// TwinCAT 3 PLC project PLC
// ProgramVersion: 3.1.4024.0
// libraries:
//   SPT Base Types, * (Beckhoff Automation LLC)
//   Tc2_Standard, * (Beckhoff Automation GmbH)
//   Tc2_System, * (Beckhoff Automation GmbH)
//   Tc3_Module, * (Beckhoff Automation GmbH)
//   Tc3_PackML_V2, * (Beckhoff Automation GmbH)
//   VisuDialogs, * (System)
// project tree:
//   DUTs/HMI/ ST_HMI_Machine.TcDUT, ST_HMI_Machine_Command.TcDUT, ST_HMI_Machine_Config.TcDUT, ST_HMI_Machine_Status.TcDUT
//   / GlobalTextList.TcGTLO, PlcTask.TcTTO, Visualization Manager.TcVMO (not stored)
//   POUs/ MAIN.TcPOU
//   VISUs/VFMs/ VFM_Machine.TcVIS, VFM_MachineControl.TcVIS, VFM_Module.TcVIS, VFM_OperatingMode.TcVIS, VFM_PackML.TcVIS, VFM_PackML_Manual.TcVIS
//   VISUs/ VIS_Main.TcVIS, VIS_TempCtrl.TcVIS
//   _Machine/00_Machine/ FB_UM_Machine.TcPOU
//   _Machine/_Components/Misc/ FB_StatFilter.TcPOU, FB_TempCtrl.TcPOU, F_TaskTime.TcPOU
//   _Machine/_Components/TempController/DUTs/ ST_HMI_TempController.TcDUT, ST_HMI_TempController_Command.TcDUT, ST_HMI_TempController_Config.TcDUT, ST_HMI_TempController_Status.TcDUT, ST_Param_TempController.TcDUT
//   _Machine/_Components/TempController/ FB_TempController.TcPOU, I_TemperatureController.TcIO
//   _Machine/_Components/TempController/VFMs/ VFM_TempController.TcVIS
// real-time tasks:
//   TASK PlcTask: cycle T#10ms, priority 20, ADS port 350

CONFIGURATION PLC
    RESOURCE PLC ON TwinCAT3
        TASK PlcTask(INTERVAL := T#10ms, PRIORITY := 20);
        PROGRAM MAIN WITH PlcTask : MAIN;
    END_RESOURCE
END_CONFIGURATION

// ---- DUTs/HMI/ST_HMI_Machine.TcDUT
TYPE ST_HMI_Machine :
STRUCT
	Command: ST_HMI_Machine_Command;
	Config: ST_HMI_Machine_Config;
	Status: ST_HMI_Machine_Status;
END_STRUCT
END_TYPE

// ---- DUTs/HMI/ST_HMI_Machine_Command.TcDUT
TYPE ST_HMI_Machine_Command :
STRUCT
	Start: BOOL;
	Stop: BOOL;
	Reset: BOOL;
	Abort: BOOL;
END_STRUCT
END_TYPE

// ---- DUTs/HMI/ST_HMI_Machine_Config.TcDUT
TYPE ST_HMI_Machine_Config :
STRUCT
END_STRUCT
END_TYPE

// ---- DUTs/HMI/ST_HMI_Machine_Status.TcDUT
TYPE ST_HMI_Machine_Status :
STRUCT
END_STRUCT
END_TYPE

// ---- _Machine/_Components/TempController/DUTs/ST_HMI_TempController.TcDUT
TYPE ST_HMI_TempController :
STRUCT
	Command: ST_HMI_TempController_Command;
	Config: ST_HMI_TempController_Config;
	Status: ST_HMI_TempController_Status;
END_STRUCT
END_TYPE

// ---- _Machine/_Components/TempController/DUTs/ST_HMI_TempController_Command.TcDUT
TYPE ST_HMI_TempController_Command :
STRUCT
	Manual: BOOL := TRUE;
	Start: BOOL;
	Stop: BOOL;
	ResetPID: BOOL;
END_STRUCT
END_TYPE

// ---- _Machine/_Components/TempController/DUTs/ST_HMI_TempController_Config.TcDUT
TYPE ST_HMI_TempController_Config :
STRUCT
	Param: ST_Param_TempController;
END_STRUCT
END_TYPE

// ---- _Machine/_Components/TempController/DUTs/ST_HMI_TempController_Status.TcDUT
TYPE ST_HMI_TempController_Status :
STRUCT
	Enabled: BOOL;
	CtrlOutput: LREAL;
	Actual: LREAL;
END_STRUCT
END_TYPE

// ---- _Machine/_Components/TempController/DUTs/ST_Param_TempController.TcDUT
TYPE ST_Param_TempController :
STRUCT
	MaxTemp: LREAL := 350.0;
	Setpoint: LREAL := 20.0;
	Range: LREAL := 10.0;
	Kp: LREAL := 1.0;
	Tn: LREAL := 0.005;
	Tv: LREAL := 0.0;
	Td: LREAL := 0.0;
END_STRUCT
END_TYPE

// ---- _Machine/_Components/TempController/I_TemperatureController.TcIO
INTERFACE I_TemperatureController

METHOD Disable
VAR_INPUT
END_VAR
END_METHOD

METHOD Enable
VAR_INPUT
END_VAR
END_METHOD

PROPERTY Enabled : bool
GET
END_GET
END_PROPERTY

END_INTERFACE

// ---- POUs/MAIN.TcPOU
(*	Sample Code Disclaimer
	All sample code provided by Beckhoff Automation LLC are for illustrative purposes only
	and are provided “as is” and without any warranties, express or implied.
	Actual implementations in applications will vary significantly.
	Beckhoff Automation LLC shall have no liability for, and does not waive any rights in relation to,
	any code samples that it provides or the use of such code samples for any purpose.
*)
PROGRAM MAIN
VAR
	Machine: FB_UM_Machine	:= (Name := 'Machine', LogStateChanges := TRUE);
	Initialized: BOOL;
END_VAR

CyclicLogic();

METHOD CyclicLogic : BOOL
VAR_INPUT
END_VAR
IF NOT Initialized THEN
    Initialized := Initialize();
    RETURN;
END_IF

Machine.CyclicLogic();
END_METHOD

METHOD Initialize : BOOL
VAR_INPUT
END_VAR
Initialize := TRUE;
END_METHOD

END_PROGRAM

// ---- _Machine/00_Machine/FB_UM_Machine.TcPOU
FUNCTION_BLOCK FB_UM_Machine EXTENDS FB_PackML_BaseModule
VAR
	// Submodules
	
	// Components
	TempController: FB_TempController	:= (Name := 'Temperature Controller');
	
	// Module Data
	// --Param
	// --Recipe
	// --HMI
	HMI: ST_HMI_Machine;
	
	// Alarms
	
	// Other I/O

	// Machine Control
	rtrigControl: R_TRIG;
	CheckAbort: BOOL;
	CheckStop: BOOL;
	
	// Miscellaneous
	
END_VAR

METHOD PROTECTED Aborted
VAR_INPUT
END_VAR
END_METHOD

METHOD PROTECTED Aborting
VAR_INPUT
END_VAR
CASE _CurrentMode OF
	E_PMLUnitMode.ePMLUnitMode_Production:
        CASE DescendantSequenceState OF
			0:
				NoStateTasksToComplete := FALSE;
				DescendantSequenceState := DescendantSequenceState + 10;
			10:
				StateTasksComplete := TRUE;
		END_CASE
		
	E_PMLUnitMode.ePMLUnitMode_Manual, E_PMLUnitMode.ePMLUnitMode_Maintenance:
        ;	
END_CASE

// Call Super
SUPER^.Aborting();
END_METHOD

METHOD PROTECTED Clearing
VAR_INPUT
END_VAR
CASE _CurrentMode OF
	E_PMLUnitMode.ePMLUnitMode_Production:
        CASE DescendantSequenceState OF
			0:
				NoStateTasksToComplete := FALSE;
				DescendantSequenceState := DescendantSequenceState + 10;
			10:
				StateTasksComplete := TRUE;
		END_CASE
		
	E_PMLUnitMode.ePMLUnitMode_Manual, E_PMLUnitMode.ePMLUnitMode_Maintenance:
        ;	
END_CASE

// Call Super
SUPER^.Clearing();
END_METHOD

METHOD PROTECTED Complete
VAR_INPUT
END_VAR
END_METHOD

//! @summary Initializes event function blocks using this module's name
METHOD PROTECTED CreateEvents

//! @description This method is called by <c>Initialize()</c> as required
// Add your event creation here

// Super call to base
SUPER^.CreateEvents();
END_METHOD

METHOD CyclicLogic
VAR_INPUT
END_VAR
IF NOT _InitComplete THEN
    _InitComplete := Initialize();
    RETURN;
END_IF

MachineControl();

SUPER^.CyclicLogic();
END_METHOD

METHOD PROTECTED Execute
VAR_INPUT
END_VAR
CASE _CurrentMode OF
	E_PMLUnitMode.ePMLUnitMode_Production:
        CASE DescendantSequenceState OF
			0:
				DescendantSequenceState := DescendantSequenceState + 10;
			10:
				;
		END_CASE
		
	E_PMLUnitMode.ePMLUnitMode_Manual, E_PMLUnitMode.ePMLUnitMode_Maintenance:
        ;	
END_CASE
END_METHOD

METHOD PROTECTED Held
VAR_INPUT
END_VAR
END_METHOD

METHOD PROTECTED Holding
VAR_INPUT
END_VAR
CASE _CurrentMode OF
	E_PMLUnitMode.ePMLUnitMode_Production:
        CASE DescendantSequenceState OF
			0:
				NoStateTasksToComplete := FALSE;
				DescendantSequenceState := DescendantSequenceState + 10;
			10:
				StateTasksComplete := TRUE;
		END_CASE
		
	E_PMLUnitMode.ePMLUnitMode_Manual, E_PMLUnitMode.ePMLUnitMode_Maintenance:
        ;	
END_CASE

// Call Super
SUPER^.Holding();
END_METHOD

METHOD PROTECTED Idle
VAR_INPUT
END_VAR
END_METHOD

//! @summary Basic module initialization logic
METHOD PROTECTED Initialize : BOOL;
VAR
	i						 : UDINT;
	varInfo					 : __SYSTEM.VAR_INFO;
	AllSubUnitsInitialized	 : BOOL := TRUE;
	AllComponentsInitialized : BOOL := TRUE;
END_VAR

//! @description This method is called by <c>CyclicLogic()</c> as required
Initialize := FALSE;
CASE DescendantSequenceState OF
    0: // Initialize
        _LogModeChanges         := FALSE;
        _LogStateChanges        := FALSE;
        DescendantSequenceState := DescendantSequenceState + 10;
	
	10: // Register Submodules
		DescendantSequenceState := DescendantSequenceState + 10;
		
    20: // Register Components
		RegisterComponent(TempController);
        DescendantSequenceState := DescendantSequenceState + 10;
		
    30: // Call the Super
        IF SUPER^.Initialize() THEN
            DescendantSequenceState := DescendantSequenceState + 10;
        END_IF
    40:
        Initialize := TRUE;
END_CASE
END_METHOD

METHOD MachineControl
VAR_INPUT
END_VAR
// Control Triggers
rtrigControl(CLK:= HMI.Command.Start XOR HMI.Command.Stop XOR HMI.Command.Reset XOR HMI.Command.Abort);

CASE CurrentState OF
	E_PMLState.ePMLState_Aborting:
		CheckAbort := FALSE;
		CheckStop := FALSE;
		
	E_PMLState.ePMLState_Aborted:
		// Wait for Reset to Clear
		IF rtrigControl.Q AND HMI.Command.Reset THEN
			ChangeState(E_PMLCommand.ePMLCommand_Clear);
		END_IF
		
	E_PMLState.ePMLState_Clearing:
		CheckAbort := TRUE;
		CheckStop := FALSE;
		
	E_PMLState.ePMLState_Stopping:
		CheckAbort := TRUE;
		CheckStop := FALSE;
		
	E_PMLState.ePMLState_Stopped:
		// Wait for Reset
		IF rtrigControl.Q AND HMI.Command.Reset THEN
			ChangeState(E_PMLCommand.ePMLCommand_Reset);
		END_IF
		
	E_PMLState.ePMLState_Resetting:
		CheckAbort := TRUE;
		CheckStop := TRUE;
	
	E_PMLState.ePMLState_Idle:
		// Wait for Start
		IF rtrigControl.Q AND HMI.Command.Start THEN
			ChangeState(E_PMLCommand.ePMLCommand_Start);
		END_IF
	
END_CASE

// Check for Abort or Stop
IF rtrigControl.Q AND HMI.Command.Abort THEN
	ChangeState(E_PMLCommand.ePMLCommand_Abort);
ELSIF rtrigControl.Q AND HMI.Command.Stop THEN
	ChangeState(E_PMLCommand.ePMLCommand_Stop);
END_IF
END_METHOD

METHOD PROTECTED Resetting
VAR_INPUT
END_VAR
CASE _CurrentMode OF
	E_PMLUnitMode.ePMLUnitMode_Production:
        CASE DescendantSequenceState OF
			0:
				NoStateTasksToComplete := FALSE;
				DescendantSequenceState := DescendantSequenceState + 10;
			10:
				StateTasksComplete := TRUE;
		END_CASE
		
	E_PMLUnitMode.ePMLUnitMode_Manual, E_PMLUnitMode.ePMLUnitMode_Maintenance:
        ;	
END_CASE

// Call Super
SUPER^.Resetting();
END_METHOD

METHOD PROTECTED Starting
VAR_INPUT
END_VAR
CASE _CurrentMode OF
	E_PMLUnitMode.ePMLUnitMode_Production:
        CASE DescendantSequenceState OF
			0:
				NoStateTasksToComplete := FALSE;
				DescendantSequenceState := DescendantSequenceState + 10;
			10:
				StateTasksComplete := TRUE;
		END_CASE
		
	E_PMLUnitMode.ePMLUnitMode_Manual, E_PMLUnitMode.ePMLUnitMode_Maintenance:
        ;	
END_CASE

// Call Super
SUPER^.Starting();
END_METHOD

METHOD PROTECTED Stopped
VAR_INPUT
END_VAR
END_METHOD

METHOD PROTECTED Stopping
VAR_INPUT
END_VAR
CASE _CurrentMode OF
	E_PMLUnitMode.ePMLUnitMode_Production:
        CASE DescendantSequenceState OF
			0:
				NoStateTasksToComplete := FALSE;
				DescendantSequenceState := DescendantSequenceState + 10;
			10:
				StateTasksComplete := TRUE;
		END_CASE
		
	E_PMLUnitMode.ePMLUnitMode_Manual, E_PMLUnitMode.ePMLUnitMode_Maintenance:
        ;	
END_CASE

// Call Super
SUPER^.Stopping();
END_METHOD

METHOD PROTECTED Suspended
VAR_INPUT
END_VAR
END_METHOD

METHOD PROTECTED Suspending
VAR_INPUT
END_VAR
CASE _CurrentMode OF
	E_PMLUnitMode.ePMLUnitMode_Production:
        CASE DescendantSequenceState OF
			0:
				NoStateTasksToComplete := FALSE;
				DescendantSequenceState := DescendantSequenceState + 10;
			10:
				StateTasksComplete := TRUE;
		END_CASE
		
	E_PMLUnitMode.ePMLUnitMode_Manual, E_PMLUnitMode.ePMLUnitMode_Maintenance:
        ;	
END_CASE

// Call Super
SUPER^.Suspending();
END_METHOD

METHOD PROTECTED Undefined
VAR_INPUT
END_VAR
END_METHOD

METHOD PROTECTED Unholding
VAR_INPUT
END_VAR
CASE _CurrentMode OF
	E_PMLUnitMode.ePMLUnitMode_Production:
        CASE DescendantSequenceState OF
			0:
				NoStateTasksToComplete := FALSE;
				DescendantSequenceState := DescendantSequenceState + 10;
			10:
				StateTasksComplete := TRUE;
		END_CASE
		
	E_PMLUnitMode.ePMLUnitMode_Manual, E_PMLUnitMode.ePMLUnitMode_Maintenance:
        ;	
END_CASE

// Call Super
SUPER^.Unholding();
END_METHOD

METHOD PROTECTED Unsuspending
VAR_INPUT
END_VAR
CASE _CurrentMode OF
	E_PMLUnitMode.ePMLUnitMode_Production:
        CASE DescendantSequenceState OF
			0:
				NoStateTasksToComplete := FALSE;
				DescendantSequenceState := DescendantSequenceState + 10;
			10:
				StateTasksComplete := TRUE;
		END_CASE
		
	E_PMLUnitMode.ePMLUnitMode_Manual, E_PMLUnitMode.ePMLUnitMode_Maintenance:
        ;	
END_CASE

// Call Super
SUPER^.Unsuspending();
END_METHOD

END_FUNCTION_BLOCK

// ---- _Machine/_Components/TempController/FB_TempController.TcPOU
(*	Sample Code Disclaimer
	All sample code provided by Beckhoff Automation LLC are for illustrative purposes only
	and are provided “as is” and without any warranties, express or implied.
	Actual implementations in applications will vary significantly.
	Beckhoff Automation LLC shall have no liability for, and does not waive any rights in relation to,
	any code samples that it provides or the use of such code samples for any purpose.
*)
FUNCTION_BLOCK FB_TempController EXTENDS FB_ComponentBase IMPLEMENTS I_TemperatureController
VAR	
	// Properties
	_Enabled: BOOL;
		
	// HMI Interface
	HMI: ST_HMI_TempController;
	
	// Hardware Inputs
	//Feedback AT %I*: INT;
	
	// Hardware Outputs
	CtrlOut AT %Q*: INT; // Scaled for HW Output

	// General
	fbTempCtrl: FB_TempCtrl;
	Setpoint: LREAL;
	Feedback: LREAL; // Scaled for HW Input
	ResetPID: BOOL;
	PID_Output: LREAL;
	EnableReq: BOOL;
	DisableReq: BOOL;
	
	// Simulation

END_VAR

VAR PERSISTENT
	Param: ST_Param_TempController;
END_VAR

METHOD CyclicLogic
VAR_INPUT
END_VAR
// Call Super
SUPER^.CyclicLogic();

IF EnableReq THEN
	_Enabled := TRUE;
	EnableReq := FALSE;
ELSIF DisableReq OR Feedback >= Param.MaxTemp THEN
	_Enabled := FALSE;	
	DisableReq := FALSE;
END_IF

// Input Scaling

// Call PID
fbTempCtrl(
	Enable:= _Enabled, 
	Setpoint:= Param.Setpoint, 
	Feedback:= Feedback, 
	MaxTemperature:= Param.MaxTemp, 
	Kp:= Param.Kp,
	Tn:= Param.Tn,
	Tv:= Param.Tv,
	Td:= Param.Td,
	ControlOutput=>PID_Output , 
);

// Method Calls
CyclicLogic_Simulation();
END_METHOD

METHOD CyclicLogic_Simulation
VAR_INPUT
END_VAR
VAR
	rLossRate: LREAL;
	rGainRate: LREAL;
END_VAR
// Simulate Heating Element
rLossRate := (Feedback - 20.0) * 6.0 / 300.0;
rGainRate := BOOL_TO_LREAL(Enabled) * 0.30 * PID_Output;
Feedback 	:= Feedback + (rGainRate - rLossRate) * fbTempCtrl.CycleTime ;
			
IF Feedback < 20.0 THEN
	Feedback := 20.0;
END_IF
END_METHOD

METHOD Disable
VAR_INPUT
END_VAR

VAR
	
END_VAR
// Disable Request
DisableReq := TRUE;
END_METHOD

METHOD Enable
VAR_INPUT
END_VAR

VAR
	
END_VAR
// Enable Request
EnableReq := TRUE;
END_METHOD

PROPERTY Enabled : BOOL
GET
Enabled := _Enabled;
END_GET
END_PROPERTY

//! @summary Provides interlocks for HMI control and updates HMI status information for this component
METHOD PROTECTED HMICommunication

//! @description This method is called cyclically by <c>CyclicLogic()</c>
// Call Super
SUPER^.HMICommunication();

Param := HMI.Config.Param;

// Manual Controls
IF HMI.Command.Manual THEN
	IF _Enabled THEN
		IF HMI.Command.Stop THEN
			Disable();
		END_IF
	ELSE
		IF HMI.Command.Start THEN
			Enable();
		END_IF
	END_IF	
END_IF

// Status Update
HMI.Status.Enabled := _Enabled;
HMI.Status.CtrlOutput := PID_Output;
HMI.Status.Actual := Feedback;
END_METHOD

//! @summary Basic component initialization logic
METHOD PROTECTED Initialize : BOOL;

//! @description This method is called by <c>CyclicLogic()</c> as required
IF fbTempCtrl.CycleTime = 0.0 THEN
	fbTempCtrl.CycleTime := F_TaskTime();
END_IF

HMI.Config.Param := Param;

//Call base class Initialize
Initialize := SUPER^.Initialize();
END_METHOD

METHOD Manual
VAR_INPUT
	ManualMode: bool;
END_VAR
HMI.Command.Manual := ManualMode;
END_METHOD

END_FUNCTION_BLOCK

// ---- _Machine/_Components/Misc/FB_TempCtrl.TcPOU
(*	Sample Code Disclaimer
	All sample code provided by Beckhoff Automation LLC are for illustrative purposes only
	and are provided “as is” and without any warranties, express or implied.
	Actual implementations in applications will vary significantly.
	Beckhoff Automation LLC shall have no liability for, and does not waive any rights in relation to,
	any code samples that it provides or the use of such code samples for any purpose.
*)
FUNCTION_BLOCK FB_TempCtrl
VAR_INPUT
	Enable: BOOL;         // Enable input for the controller
	CycleTime: LREAL;     // Time between controller calculations
	Setpoint: LREAL;      // Desired temperature setpoint
	Feedback: LREAL;      // Current temperature feedback
	MaxTemperature: LREAL; // Maximum allowable temperature
	Kp: LREAL;            // Proportional gain
	Tn: LREAL;            // Integral time constant
	Tv: LREAL;            // Derivative time constant
	Td: LREAL;            // Derivative time delay
END_VAR
VAR_OUTPUT
	Enabled: BOOL;        // Output indicating if the controller is enabled
	ControlOutput: LREAL;  // Control output between 0-100%

END_VAR

VAR
	Integral: LREAL := 0.0;
	Proportional: LREAL;
	Derivative: LREAL;
	FeedBackError: LREAL;     // Error between setpoint and feedback
	PrevError: LREAL := 0.0; // Previous error value for derivative calculation
END_VAR

    // Check if the controller is enabled
    IF Enable THEN
        // Calculate the error
        FeedBackError := Setpoint - Feedback;
        
        // Proportional term
        Proportional := Kp * FeedBackError;
        
        // Integral term with anti-reset windup
		IF Tn > 0.0 THEN
			Integral := Integral + (Kp / Tn) * FeedBackError * CycleTime;
		ELSE
			Integral := 0.0; 
		END_IF
        
        IF Integral > MaxTemperature THEN
            Integral := MaxTemperature; // Anti-reset windup
        ELSIF Integral < 0.0 THEN
            Integral := 0.0; // Anti-reset windup
        END_IF

        // Derivative term
        Derivative := -Kp * Tv * (FeedBackError - PrevError) / (Td + CycleTime);
        
        // Calculate control output
        ControlOutput := Proportional + Integral + Derivative;
        
        // Clamp control output to the range [0, 100]
        IF ControlOutput > 100.0 THEN
            ControlOutput := 100.0;
        ELSIF ControlOutput < 0.0 THEN
            ControlOutput := 0.0;
        END_IF
        
        // Update previous error for next iteration
        PrevError := FeedBackError;
        
        // Set the Enabled output to TRUE
        Enabled := TRUE;
        
    ELSE
        // If the controller is disabled, set outputs to default values
        ControlOutput := 0.0;
        Integral := 0.0;
        PrevError := 0.0;
        
        // Set the Enabled output to FALSE
        Enabled := FALSE;
    END_IF

END_FUNCTION_BLOCK

// ---- _Machine/_Components/Misc/F_TaskTime.TcPOU
(*	Sample Code Disclaimer
	All sample code provided by Beckhoff Automation LLC are for illustrative purposes only
	and are provided “as is” and without any warranties, express or implied.
	Actual implementations in applications will vary significantly.
	Beckhoff Automation LLC shall have no liability for, and does not waive any rights in relation to,
	any code samples that it provides or the use of such code samples for any purpose.
*)
FUNCTION F_TaskTime : LREAL
VAR
END_VAR

// Get Current Task Scan Time and convert to seconds
F_TaskTime := UDINT_TO_LREAL(_TaskInfo[GETCURTASKINDEXEX()].CycleTime) / 10000000.0;

END_FUNCTION

// ---- _Machine/_Components/Misc/FB_StatFilter.TcPOU
(*	Sample Code Disclaimer
	All sample code provided by Beckhoff Automation LLC are for illustrative purposes only
	and are provided “as is” and without any warranties, express or implied.
	Actual implementations in applications will vary significantly.
	Beckhoff Automation LLC shall have no liability for, and does not waive any rights in relation to,
	any code samples that it provides or the use of such code samples for any purpose.
*)
FUNCTION_BLOCK FB_StatFilter
VAR
	// Properties
	_Weight: UDINT := 1;
	_Count: UDINT;
	_Valid: BOOL;
	_LastValue: LREAL;
	_Minimum: LREAL;
	_Maximum: LREAL;
	_Avg: LREAL;
	_RMS: LREAL;
	_StdDev: LREAL;
	_StdErr: LREAL;
	
	rCount: LREAL;
	nIter: INT;
END_VAR

PROPERTY Avg : LREAL
GET
Avg := _Avg;
END_GET
END_PROPERTY

PROPERTY Count : UDINT
GET
Count := _Count;
END_GET
END_PROPERTY

PROPERTY LastValue : LREAL
GET
LastValue := _LastValue;
END_GET
END_PROPERTY

PROPERTY Maximum : LREAL
GET
Maximum := _Maximum;
END_GET
END_PROPERTY

PROPERTY Minimum : LREAL
GET
Minimum := _Minimum;
END_GET
END_PROPERTY

METHOD Reset : BOOL
VAR_INPUT
END_VAR

VAR
	
END_VAR
// Reset Stats
_Valid := FALSE;
_Count := 0;
_Minimum := 0;
_Maximum := 0;
_Avg := 0.0;
_StdDev := 0.0;
_StdErr := 0.0;
END_METHOD

PROPERTY RMS : LREAL
GET
RMS := _RMS;
END_GET
END_PROPERTY

METHOD Sample : BOOL
VAR_INPUT
	Value: lreal;
END_VAR
_Count := _Count +1;
IF _Count < _Weight OR _Weight = 0 THEN
	rCount := UDINT_TO_REAL(_Count);
ELSE
	_Valid := TRUE;
	rCount := UDINT_TO_REAL(_Weight);
END_IF

IF rCount > 0.0 THEN
	IF rCount = 1 OR Value < _Minimum THEN
		_Minimum := Value;
	END_IF
	
	IF rCount = 1 OR Value > _Maximum THEN
		_Maximum := Value;
	END_IF
	
	_Avg := (Value + _Avg * (rCount-1.0))/ rCount;
	_RMS := SQRT(  ( EXPT(Value,2)        + (rCount-1.0)*EXPT(_RMS,2)    ) / rCount  );
	_StdDev := SQRT(  ( EXPT(Value-_Avg,2) + (rCount-1.0)*EXPT(_StdDev,2) ) / rCount );
	_StdErr := _StdDev/ SQRT(rCount);

END_IF

_LastValue := Value;
END_METHOD

PROPERTY StdDev : LREAL
GET
StdDev := _StdDev;
END_GET
END_PROPERTY

PROPERTY StdErr : LREAL
GET
StdErr := _StdErr;
END_GET
END_PROPERTY

PROPERTY Valid : BOOL
GET
Valid := _Valid;
END_GET
END_PROPERTY

PROPERTY Weight : UDINT
GET
Weight := _Weight;
END_GET
SET
IF Weight <> _Weight THEN
	_Valid := FALSE;
	_Count := 0;
	_Minimum := 0;
	_Maximum := 0;
	_Avg := 0.0;
	_StdDev := 0.0;
	_StdErr := 0.0;
END_IF

_Weight := Weight;
END_SET
END_PROPERTY

END_FUNCTION_BLOCK

// ---- GlobalTextList.TcGTLO
TEXTLIST GlobalTextList
  672 = '%3.1f %%'
  685 = '%s'
  680 = 'Abort'
  11 = 'Aborted'
  86 = 'Aborting'
  452 = 'Clear'
  467 = 'Clearing'
  754 = 'Complete'
  302 = 'Completing'
  663 = 'Execute'
  51 = 'Held'
  744 = 'Hold'
  369 = 'Holding'
  236 = 'I'
  342 = 'Idle'
  46 = 'Maintenance'
  904 = 'Manual'
  820 = 'O'
  929 = 'Production'
  263 = 'PV: %3.1f'
  799 = 'R'
  181 = 'Reset'
  123 = 'Resetting'
  639 = 'SC'
  77 = 'Start'
  888 = 'Starting'
  516 = 'State: %s'
  828 = 'Stop'
  796 = 'Stopped'
  161 = 'Stopping'
  806 = 'Suspend'
  623 = 'Suspended'
  229 = 'Suspending'
  304 = 'SV: %3.1f'
  124 = 'Temp Controller'
  782 = 'Un-Hold'
  466 = 'Un-Holding'
  901 = 'Un-Suspend'
  254 = 'Un-Suspending'
  197 = 'Unhold'
  832 = 'Unsuspend'
END_TEXTLIST

// ---- VISUs/VFMs/VFM_Machine.TcVIS
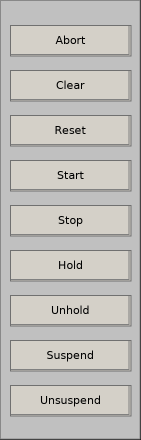
VISUALIZATION VFM_Machine  // 141x440
VAR_IN_OUT
	HMI : ST_PackMLBaseModule_HMI;
END_VAR
    Rectangle (0,0 141x440)
    Button (10,25 121x31), "Abort"
        OnMouseClick: execute { HMI.Command.State := E_PMLCommand.ePMLCommand_Abort; }
    Button (10,70 121x31), "Clear"
        OnMouseClick: execute { HMI.Command.State := E_PMLCommand.ePMLCommand_Clear; }
    Button (10,115 121x31), "Reset"
        OnMouseClick: execute { HMI.Command.State := E_PMLCommand.ePMLCommand_Reset; }
    Button (10,160 121x31), "Start"
        OnMouseClick: execute { HMI.Command.State := E_PMLCommand.ePMLCommand_Start; }
    Button (10,205 121x31), "Stop"
        OnMouseClick: execute { HMI.Command.State := E_PMLCommand.ePMLCommand_Stop; }
    Button (10,250 121x31), "Hold"
        OnMouseClick: execute { HMI.Command.State := E_PMLCommand.ePMLCommand_Hold; }
    Button (10,295 121x31), "Unhold"
        OnMouseClick: execute { HMI.Command.State := E_PMLCommand.ePMLCommand_Unhold; }
    Button (10,340 121x31), "Suspend"
        OnMouseClick: execute { HMI.Command.State := E_PMLCommand.ePMLCommand_Suspend; }
    Button (10,385 121x31), "Unsuspend"
        OnMouseClick: execute { HMI.Command.State := E_PMLCommand.ePMLCommand_Unsuspend; }
END_VISUALIZATION

// ---- VISUs/VFMs/VFM_MachineControl.TcVIS
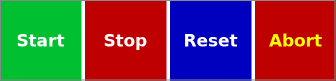
VISUALIZATION VFM_MachineControl  // 336x81
VAR_IN_OUT
	HMI: ST_HMI_Machine;
END_VAR
    Rectangle (0,0 81x81), "Start"
        tap HMI.Command.Start
    Rectangle (85,0 81x81), "Stop"
        tap HMI.Command.Stop
    Rectangle (170,0 81x81), "Reset"
        tap HMI.Command.Reset
    Rectangle (255,0 81x81), "Abort"
        toggle HMI.Command.Abort
END_VISUALIZATION

// ---- VISUs/VFMs/VFM_Module.TcVIS
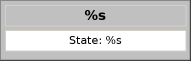
VISUALIZATION VFM_Module  // 191x61
VAR_IN_OUT
	HMI : ST_PackMLBaseModule_HMI;
END_VAR
    Rectangle (0,0 191x61)
    Textfield (5,5 181x21), "%s", text variable: HMI.Config.Name
    Textfield (5,30 181x21), "State: %s", text variable: HMI.Status.State
END_VISUALIZATION

// ---- VISUs/VFMs/VFM_OperatingMode.TcVIS
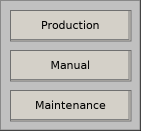
VISUALIZATION VFM_OperatingMode  // 141x131
VAR_IN_OUT
	HMI : ST_PackMLBaseModule_HMI;
END_VAR
    Rectangle (0,0 141x131)
    Button (10,10 121x31), "Production", colour toggle: HMI.Status.Mode = E_PMLUnitMode.ePMLUnitMode_Production
        OnMouseClick: execute { HMI.Command.Mode := E_PMLUnitMode.ePMLUnitMode_Production; }
    Button (10,50 121x31), "Manual", colour toggle: HMI.Status.Mode = E_PMLUnitMode.ePMLUnitMode_Manual
        OnMouseClick: execute { HMI.Command.Mode := E_PMLUnitMode.ePMLUnitMode_Manual; }
    Button (10,90 121x31), "Maintenance", colour toggle: HMI.Status.Mode = E_PMLUnitMode.ePMLUnitMode_Maintenance
        OnMouseClick: execute { HMI.Command.Mode := E_PMLUnitMode.ePMLUnitMode_Maintenance; }
END_VISUALIZATION

// ---- VISUs/VFMs/VFM_PackML.TcVIS
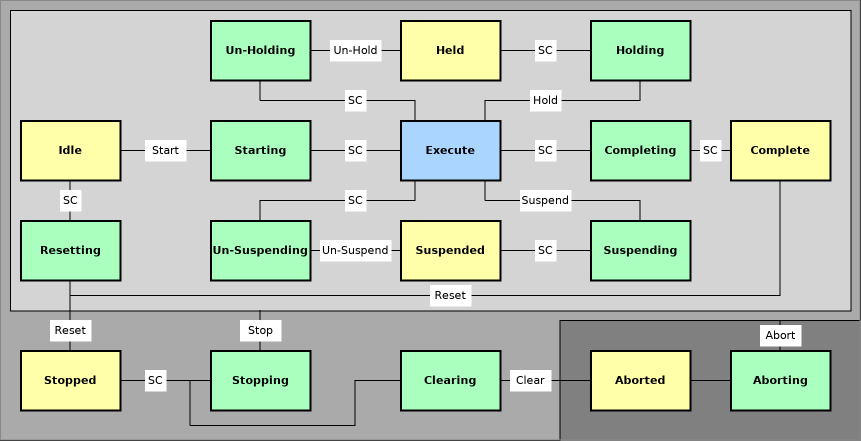
VISUALIZATION VFM_PackML  // 861x441
VAR_IN_OUT
	HMI : ST_PackMLBaseModule_HMI;
END_VAR
    Rectangle (560,320 301x121)
    Rectangle (10,10 841x301)
    Rectangle (590,350 101x61), "Aborted", colour toggle: HMI.Status.State = Tc3_PackML_V2.E_PMLState.ePMLState_Aborted
    Rectangle (400,350 101x61), "Clearing", colour toggle: HMI.Status.State = Tc3_PackML_V2.E_PMLState.ePMLState_Clearing
    Rectangle (210,350 101x61), "Stopping", colour toggle: HMI.Status.State = Tc3_PackML_V2.E_PMLState.ePMLState_Stopping
    Rectangle (20,350 101x61), "Stopped", colour toggle: HMI.Status.State = Tc3_PackML_V2.E_PMLState.ePMLState_Stopped
    Rectangle (20,220 101x61), "Resetting", colour toggle: HMI.Status.State = Tc3_PackML_V2.E_PMLState.ePMLState_Resetting
    Rectangle (20,120 101x61), "Idle", colour toggle: HMI.Status.State = Tc3_PackML_V2.E_PMLState.ePMLState_Idle
    Rectangle (210,120 101x61), "Starting", colour toggle: HMI.Status.State = Tc3_PackML_V2.E_PMLState.ePMLState_Starting
    Rectangle (400,120 101x61), "Execute", colour toggle: HMI.Status.State = Tc3_PackML_V2.E_PMLState.ePMLState_Execute
    Rectangle (590,20 101x61), "Holding", colour toggle: HMI.Status.State = Tc3_PackML_V2.E_PMLState.ePMLState_Holding
    Rectangle (400,20 101x61), "Held", colour toggle: HMI.Status.State = Tc3_PackML_V2.E_PMLState.ePMLState_Held
    Rectangle (210,20 101x61), "Un-Holding", colour toggle: HMI.Status.State = Tc3_PackML_V2.E_PMLState.ePMLState_Unholding
    Rectangle (590,220 101x61), "Suspending", colour toggle: HMI.Status.State = Tc3_PackML_V2.E_PMLState.ePMLState_Suspending
    Rectangle (400,220 101x61), "Suspended", colour toggle: HMI.Status.State = Tc3_PackML_V2.E_PMLState.ePMLState_Suspended
    Rectangle (210,220 101x61), "Un-Suspending", colour toggle: HMI.Status.State = Tc3_PackML_V2.E_PMLState.ePMLState_Unsuspending
    Rectangle (590,120 101x61), "Completing", colour toggle: HMI.Status.State = Tc3_PackML_V2.E_PMLState.ePMLState_Completing
    Rectangle (730,120 101x61), "Complete", colour toggle: HMI.Status.State = Tc3_PackML_V2.E_PMLState.ePMLState_Complete
    Rectangle (730,350 101x61), "Aborting", colour toggle: HMI.Status.State = Tc3_PackML_V2.E_PMLState.ePMLState_Aborting
    Line (0,0) (860,0)
    Line (860,0) (860,320)
    Line (560,320) (860,320)
    Line (560,440) (560,320)
    Line (0,440) (560,440)
    Line (0,440) (0,0)
    Line (780,350) (780,320)
    Line (690,380) (730,380)
    Line (355,380) (400,380)
    Line (500,380) (590,380)
    Line (355,425) (355,380)
    Line (190,425) (355,425)
    Line (260,350) (260,310)
    Line (120,380) (210,380)
    Line (310,250) (400,250)
    Line (500,250) (590,250)
    Line (500,50) (590,50)
    Line (310,50) (400,50)
    Line (120,150) (210,150)
    Line (310,150) (400,150)
    Line (500,150) (590,150)
    Line (690,150) (730,150)
    Line (70,295) (780,295)
    Line (190,425) (190,380)
    Line (70,350) (70,280)
    Line (780,295) (780,180)
    Line (70,220) (70,180)
    Line (485,100) (640,100)
    Line (640,100) (640,80)
    Line (485,120) (485,100)
    Line (640,220) (640,200)
    Line (485,200) (640,200)
    Line (485,200) (485,180)
    Line (260,100) (260,80)
    Line (415,120) (415,100)
    Line (260,100) (415,100)
    Line (260,220) (260,200)
    Line (260,200) (415,200)
    Line (415,200) (415,180)
    Rectangle (760,325 41x21), "Abort"
    Rectangle (50,320 41x21), "Reset"
    Rectangle (510,370 41x21), "Clear"
    Rectangle (240,320 41x21), "Stop"
    Rectangle (145,370 21x21), "SC"
    Rectangle (60,190 21x21), "SC"
    Rectangle (345,140 21x21), "SC"
    Rectangle (535,140 21x21), "SC"
    Rectangle (535,40 21x21), "SC"
    Rectangle (700,140 21x21), "SC"
    Rectangle (535,240 21x21), "SC"
    Rectangle (345,190 21x21), "SC"
    Rectangle (345,90 21x21), "SC"
    Rectangle (530,90 31x21), "Hold"
    Rectangle (520,190 51x21), "Suspend"
    Rectangle (320,240 71x21), "Un-Suspend"
    Rectangle (330,40 51x21), "Un-Hold"
    Rectangle (430,285 41x21), "Reset"
    Rectangle (145,140 41x21), "Start"
END_VISUALIZATION

// ---- VISUs/VFMs/VFM_PackML_Manual.TcVIS
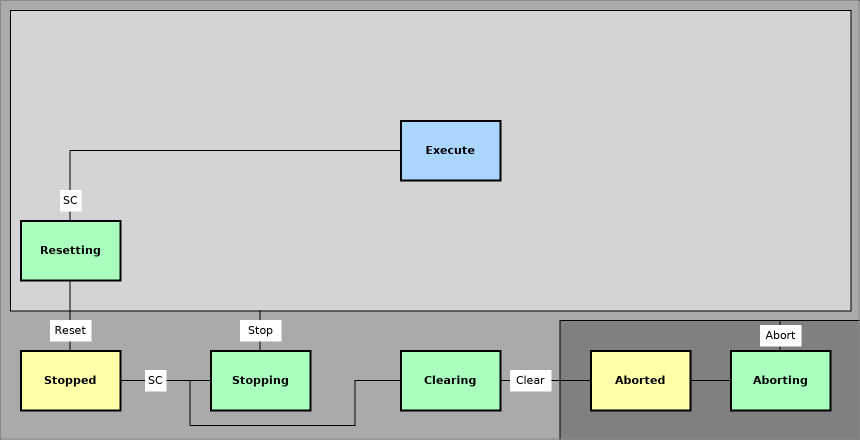
VISUALIZATION VFM_PackML_Manual  // 860x440
VAR_IN_OUT
	HMI : ST_PackMLBaseModule_HMI;
END_VAR
    Rectangle (560,320 301x121)
    Rectangle (10,10 841x301)
    Rectangle (590,350 101x61), "Aborted", colour toggle: HMI.Status.State = Tc3_PackML_V2.E_PMLState.ePMLState_Aborted
    Rectangle (400,350 101x61), "Clearing", colour toggle: HMI.Status.State = Tc3_PackML_V2.E_PMLState.ePMLState_Clearing
    Rectangle (210,350 101x61), "Stopping", colour toggle: HMI.Status.State = Tc3_PackML_V2.E_PMLState.ePMLState_Stopping
    Rectangle (20,350 101x61), "Stopped", colour toggle: HMI.Status.State = Tc3_PackML_V2.E_PMLState.ePMLState_Stopped
    Rectangle (20,220 101x61), "Resetting", colour toggle: HMI.Status.State = Tc3_PackML_V2.E_PMLState.ePMLState_Resetting
    Rectangle (400,120 101x61), "Execute", colour toggle: HMI.Status.State = Tc3_PackML_V2.E_PMLState.ePMLState_Execute
    Rectangle (730,350 101x61), "Aborting", colour toggle: HMI.Status.State = Tc3_PackML_V2.E_PMLState.ePMLState_Aborting
    Line (0,0) (860,0)
    Line (860,0) (860,320)
    Line (560,320) (860,320)
    Line (560,440) (560,320)
    Line (0,440) (560,440)
    Line (0,440) (0,0)
    Line (780,350) (780,320)
    Line (690,380) (730,380)
    Line (355,380) (400,380)
    Line (500,380) (590,380)
    Line (355,425) (355,380)
    Line (190,425) (355,425)
    Line (260,350) (260,310)
    Line (120,380) (210,380)
    Line (70,150) (400,150)
    Line (190,425) (190,380)
    Line (70,350) (70,280)
    Line (70,220) (70,150)
    Rectangle (760,325 41x21), "Abort"
    Rectangle (50,320 41x21), "Reset"
    Rectangle (510,370 41x21), "Clear"
    Rectangle (240,320 41x21), "Stop"
    Rectangle (145,370 21x21), "SC"
    Rectangle (60,190 21x21), "SC"
END_VISUALIZATION

// ---- VISUs/VIS_Main.TcVIS
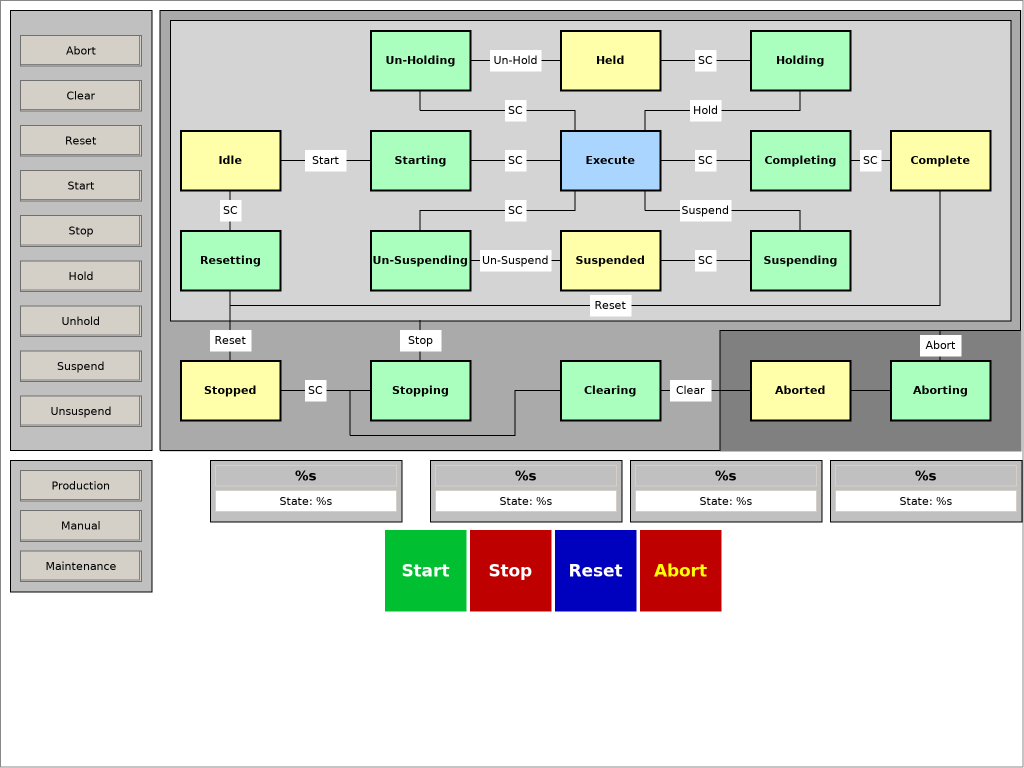
VISUALIZATION VIS_Main  // 1024x768
    Frame (160,10 861x441)
        shows VFM_PackML(HMI := MAIN.Machine.PackMLBaseModule_HMI)
    Frame (385,530 336x81)
        shows VFM_MachineControl(HMI := MAIN.Machine.HMI)
    Frame (10,10 142x441)
        shows VFM_Machine(HMI := MAIN.Machine.PackMLBaseModule_HMI)
    Frame (10,460 142x132)
        shows VFM_OperatingMode(HMI := MAIN.Machine.PackMLBaseModule_HMI)
    Frame (210,460 192x62)
        shows VFM_Module(HMI := MAIN.Machine.PackMLBaseModule_HMI)
    Frame (430,460 192x62)
        shows VFM_Module(HMI := MAIN.Machine.EM_Infeed.PackMLBaseModule_HMI)
    Frame (630,460 192x62)
        shows VFM_Module(HMI := MAIN.Machine.EM_Work.PackMLBaseModule_HMI)
    Frame (830,460 192x62)
        shows VFM_Module(HMI := MAIN.Machine.EM_Outfeed.PackMLBaseModule_HMI)
END_VISUALIZATION

// ---- VISUs/VIS_TempCtrl.TcVIS
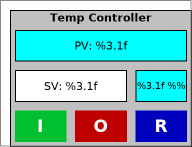
VISUALIZATION VIS_TempCtrl  // 192x147
    Frame (10,10 182x137)
        shows VFM_TempController(HMI := MAIN.Machine.TempController.HMI)
END_VISUALIZATION

// ---- _Machine/_Components/TempController/VFMs/VFM_TempController.TcVIS
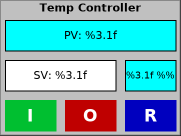
VISUALIZATION VFM_TempController  // 181x136
VAR_IN_OUT
	HMI: ST_HMI_TempController;
END_VAR
    Rectangle (0,0 181x136), "Temp Controller"
    Rectangle (5,20 171x31), "PV: %3.1f", text variable: HMI.Status.Actual, input disabled if: NOT HMI.Status.Enabled
    Rectangle (5,60 111x31), "SV: %3.1f", text variable: HMI.Config.Param.Setpoint, input disabled if: NOT HMI.Status.Enabled
        OnMouseClick: write the text variable via Default
    Rectangle (5,100 51x31), "I", input disabled if: NOT HMI.Command.Manual
        tap HMI.Command.Start
    Rectangle (125,100 51x31), "R", input disabled if: NOT HMI.Command.Manual
        tap HMI.Command.ResetPID
    Rectangle (65,100 51x31), "O", input disabled if: NOT HMI.Command.Manual
        tap HMI.Command.Stop
    Rectangle (125,60 51x31), "%3.1f %%", text variable: HMI.Status.CtrlOutput, input disabled if: NOT HMI.Status.Enabled
END_VISUALIZATION
